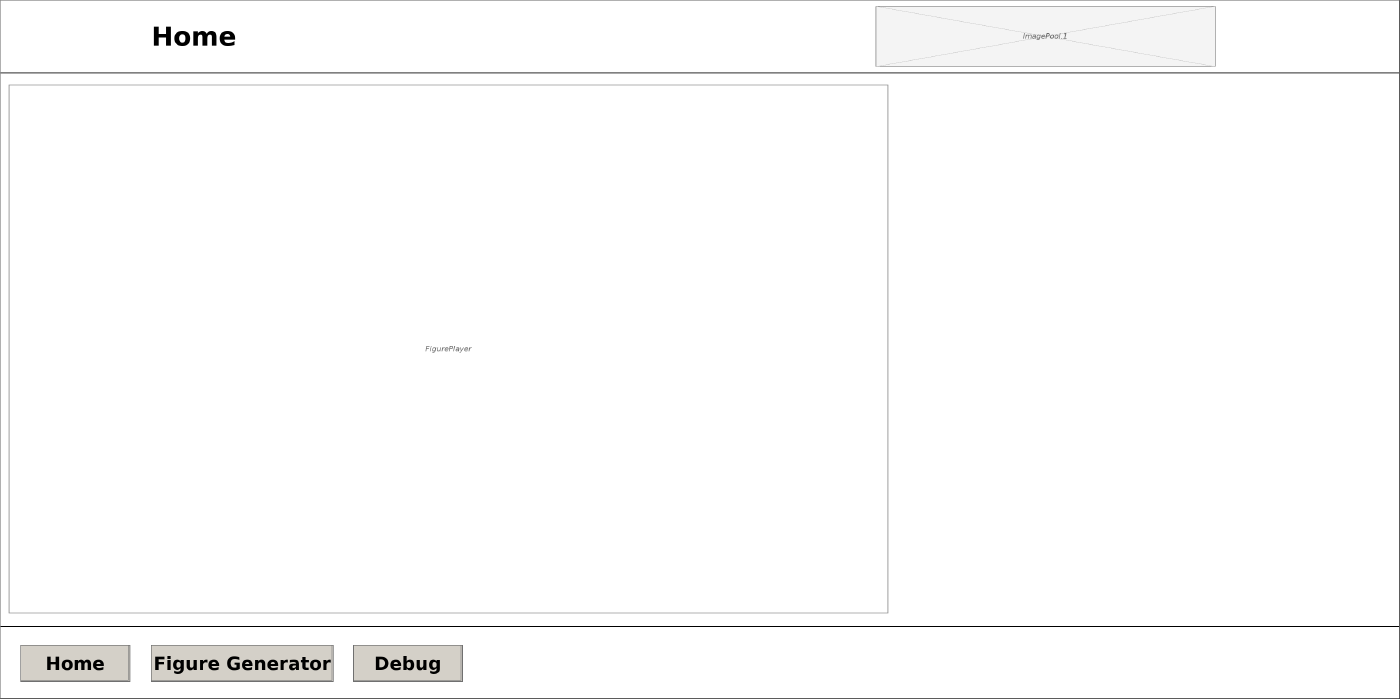
VISUALIZATION Home  // 1919x959
    Rectangle (0,0 1919x910)
    Rectangle (0,0 1919x100)
    Rectangle (0,859 1919x100)
    Button (28,885 150x50), "Home"
    Label (191,25 150x50), "Home"
    Image (1200,8 466x83), image: ImagePool.1
    Button (207,885 250x50), "Figure Generator"
        OnMouseClick: change screen: FigureGenerator1
    Button (484,885 150x50), "Debug"
        OnMouseClick: change screen: Debug
    Frame (12,116 1205x725)
        shows FigurePlayer()
END_VISUALIZATION

(* stored: Version 1.1.0.1, ProductVersion 3.1.4024.12
   Visu Home: Id {cc11e0fb-8e99-4dd4-87a1-19e1efca5965} *)
